// TwinCAT 3 PLC project PLC
// ProgramVersion: 3.1.4026.23
// libraries:
//   Tc2_EtherCAT, * (Beckhoff Automation GmbH)
//   Tc2_Standard, * (Beckhoff Automation GmbH)
//   Tc2_System, * (Beckhoff Automation GmbH)
// project tree:
//   / PlcTask.TcTTO
//   POUs/ F_ConsumeTime.TcPOU (not stored), MAIN.TcPOU
// real-time tasks:
//   TASK PlcTask: cycle T#10ms, priority 20, ADS port 350
//   TASK cppTask: cycle T#10ms, priority 15, ADS port 351
// variable links:
//   PLC/PLC 1 <-> PLC/PLC 2
//     PlcTask Inputs/MAIN.In_1 <-> PlcTask Outputs/MAIN.Counter
//     PlcTask Outputs/MAIN.Counter <-> PlcTask Inputs/MAIN.In_1
//   PLC/PLC 1 <-> PLC/PLC 3
//     PlcTask Inputs/MAIN.In_2 <-> PlcTask Outputs/MAIN.Counter
//     PlcTask Outputs/MAIN.Counter <-> PlcTask Inputs/MAIN.In_1
//   PLC/PLC 2 <-> PLC/PLC 3
//     PlcTask Inputs/MAIN.In_2 <-> PlcTask Outputs/MAIN.Counter
//     PlcTask Outputs/MAIN.Counter <-> PlcTask Inputs/MAIN.In_2
//   cpp/Obj1 <-> cpp/Obj2
//     Inputs/Counter1 <-> Outputs/ToX
//     Outputs/ToX <-> Inputs/Counter1
//   cpp/Obj1 <-> cpp/Obj3
//     Inputs/Counter2 <-> Outputs/ToX
//     Outputs/ToX <-> Inputs/Counter1
//   cpp/Obj2 <-> cpp/Obj3
//     Inputs/Counter2 <-> Outputs/ToX
//     Outputs/ToX <-> Inputs/Counter2

CONFIGURATION PLC
    RESOURCE PLC ON TwinCAT3
        TASK PlcTask(INTERVAL := T#10ms, PRIORITY := 20);
        PROGRAM MAIN WITH PlcTask : MAIN;
    END_RESOURCE
END_CONFIGURATION

// ---- POUs/MAIN.TcPOU
PROGRAM MAIN
VAR
	Counter AT %Q* : UDINT;
	In_1	AT %I* : UDINT;
	In_2	AT %I* : UDINT;
	
	{attribute 'TcInitSymbol'}
	TimeToConsume :UDINT:=10;
END_VAR

F_ConsumeTime(TimeToConsume);
Counter := (Counter + 1) MOD 200;

END_PROGRAM
